FUNCTION_BLOCK fbSimFCV
VAR_INPUT
	CmdSpOut : REAL;
END_VAR
VAR_OUTPUT
	ActPos : REAL;
END_VAR
VAR
	tonStepInc : TON;
	tStep : TIME := T#1MS;
	rStep : REAL := 1;
END_VAR

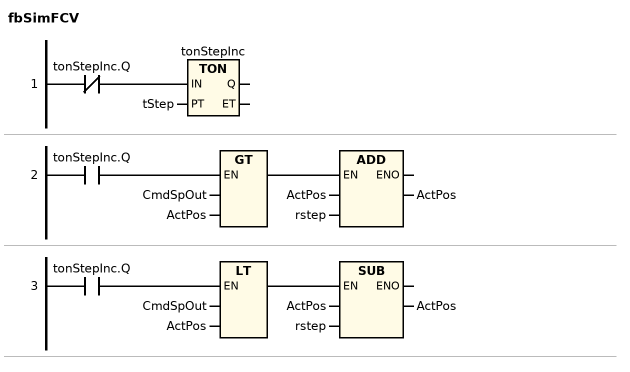
// NETWORK 1
tonStepInc(IN := NOT tonStepInc.Q, PT := tStep); // TON

// NETWORK 2
IF tonStepInc.Q AND CmdSpOut > ActPos THEN ActPos := ActPos + rstep; END_IF

// NETWORK 3
IF tonStepInc.Q AND CmdSpOut < ActPos THEN ActPos := ActPos - rstep; END_IF

END_FUNCTION_BLOCK

(* stored: Version 1.1.0.1, ProductVersion 3.1.4022.17
   POU fbSimFCV: Id {c2b92812-c33c-4281-a9c1-4593babffbfd}, SpecialFunc None *)
